Staubli VAL3: NUM.pjx

--- NUM.pjx ---
Parameters version=s7.5 stackSize=5000 millimeterUnit=true
Program file=condition.pgx
Program file=find.pgx
Program file=get.pgx
Program file=getSize.pgx
Program file=getType.pgx
Program file=isActive.pgx
Program file=load.pgx
Program file=make_if.pgx
Program file=make_NUM.pgx
Program file=onEdit.pgx
Program file=onInsert.pgx
Program file=onProgEnd.pgx
Program file=onRun.pgx
Program file=onStart.pgx
Program file=onStop.pgx
Program file=selectType.pgx
Program file=set.pgx
Program file=setValue.pgx
Data file=NUM.dtx
Library alias=use path=Disk://kernel/userPage/userPage.pjx
Library alias=cycleStatus path=Disk://cycleStatus/cycleStatus.pjx
Library alias=language path=Disk://kernel/language/language.pjx
Library alias=saveInOut path=Disk://saveInputOutput/saveInputOutput.pjx
Type name=aioItem path=Disk://kernel/template/aioItem/aioItem.pjx
Type name=countItem path=Disk://kernel/template/countItem/countItem.pjx

--- NUM.dtx ---
public string sItems
num nIndex
string sMessage
num nMode

--- condition.pgx ---
public program condition(num x_nOperator, num x_nValue, string x_sItem, bool& x_bResult)
begin
  // operator
  // <> >= > < <= ==
  x_bResult=false
  //
  switch x_nOperator
    case 0
      // <>
      if isDefined(saveInOut:cCount[x_sItem])
        x_bResult=(saveInOut:cCount[x_sItem].nCount!=x_nValue)
      elseIf isDefined(saveInOut:aCount[x_sItem])
        x_bResult=(aioGet(saveInOut:aCount[x_sItem].aAio)!=x_nValue)
      endIf
    break
    case 1
      // >=
      if isDefined(saveInOut:cCount[x_sItem])
        x_bResult=(saveInOut:cCount[x_sItem].nCount>=x_nValue)
      elseIf isDefined(saveInOut:aCount[x_sItem])
        x_bResult=(aioGet(saveInOut:aCount[x_sItem].aAio)>=x_nValue)
      endIf
    break
    case 2
      // >
      if isDefined(saveInOut:cCount[x_sItem])
        x_bResult=(saveInOut:cCount[x_sItem].nCount>x_nValue)
      elseIf isDefined(saveInOut:aCount[x_sItem])
        x_bResult=(aioGet(saveInOut:aCount[x_sItem].aAio)>x_nValue)
      endIf
    break
    case 3
      // <
      if isDefined(saveInOut:cCount[x_sItem])
        x_bResult=(saveInOut:cCount[x_sItem].nCount<x_nValue)
      elseIf isDefined(saveInOut:aCount[x_sItem])
        x_bResult=(aioGet(saveInOut:aCount[x_sItem].aAio)<x_nValue)
      endIf
    break
    case 4
      // <=
      if isDefined(saveInOut:cCount[x_sItem])
        x_bResult=(saveInOut:cCount[x_sItem].nCount<=x_nValue)
      elseIf isDefined(saveInOut:aCount[x_sItem])
        x_bResult=(aioGet(saveInOut:aCount[x_sItem].aAio)<=x_nValue)
      endIf
    break
    case 5
      // ==
      if isDefined(saveInOut:cCount[x_sItem])
        x_bResult=(saveInOut:cCount[x_sItem].nCount==x_nValue)
      elseIf isDefined(saveInOut:aCount[x_sItem])
        x_bResult=(aioGet(saveInOut:aCount[x_sItem].aAio)==x_nValue)
      endIf
    break
  endSwitch
end

--- find.pgx ---
public program find(string& x_sItem[], bool& x_bFound[])
  local num l_nIndex
  local num l_nOperator
  local num l_nValue
  local string l_sItem[2]
begin
  // REMOVE THE COUNT
  x_sItem=right(x_sItem,len(x_sItem)-len("NUM "))
  // look inside
  x_bFound=isDefined(saveInOut:cCount[x_sItem])
  if !x_bFound
    x_bFound=isDefined(saveInOut:aCount[x_sItem])
  endIf
end

--- isActive.pgx ---
public program isActive(bool& x_bActive, string x_sItem)
begin
  // check it
  if isDefined(saveInOut:cCount[x_sItem])
    x_bActive=saveInOut:cCount[x_sItem].bActive
  elseIf isDefined(saveInOut:aCount[x_sItem])
    x_bActive=(ioStatus(saveInOut:aCount[x_sItem].aAio)>=0)
  else
    // not found
    // toDO
    popUpMsg("value not found: "+x_sItem)
    x_sItem=""
  endIf
end

--- make_if.pgx ---
program make_if(string& x_sItem)
  local string l_sMessage
  local num i
  local num l_nValue
  local string l_sEmpty
  local string l_sItem
  local num l_nSizeList
  local string l_sEvent
  local bool l_bActive
  local string l_sItemList
  local num l_nKey
  local num l_nIndex
  local string l_sButton[2]
  local bool l_bYes
begin
  //
  cls()
  // Select the operator
  call language:message(l_sMessage,110)
  call use:questionDialog(l_sMessage,saveInOut:sCondition,i)
  //
  // != >= > < <= ==
  // compose the istruction
  if i>=1 and i<=size(saveInOut:sCondition)
    x_sItem=x_sItem+saveInOut:sCondition[i-1]
  else
    // escape
    x_sItem=""
    return
  endIf
  // modify the actual item
  call use:type(2,12,x_sItem)
  // insert a value
  call language:message(l_sMessage,112)
  // get the yes_no button Key
  call language:getYesNo(l_sButton)
  // ask the question
  call use:yes_no(l_sMessage,l_sButton,l_bYes)
  // check it
  if l_bYes
    //
    // reuse the operator
    //
    call saveInOut:getSize_num(l_nSizeList)
    call getType(l_sItem)
    call use:setSizeList(21,0,17,10)
    call use:listcreate(l_sItem)
    // insert in the list
    for i=0 to l_nSizeList-1
      call saveInOut:get_num(l_sItemList,i)
      call isActive(l_bActive,l_sItemList)
      if l_bActive
        call use:listadd(l_sItemList)
      endIf
    endFor
    call use:listredraw(0)
    do
      // get the key
      l_nKey=get()
      // get one input from the list
      call use:listevent(l_nKey,l_nIndex,l_sEvent)
      if l_nKey==255
        return
      endIf
    until l_nKey==270
    // check if an item has been selected
    if l_sEvent==""
      x_sItem=""
      return
    else
      x_sItem=x_sItem+"NUM "+ l_sEvent
    endIf
  else
    // use a value
    call use:changeValue(l_nValue,-10000,10000,2+len(x_sItem),12,l_sEmpty)
    x_sItem=x_sItem+toString("",l_nValue)
  endIf
  // validate
  if use:bUseEscape
    x_sItem=""
  endIf
end

--- make_NUM.pgx ---
program make_NUM(string& x_sItem)
  local string l_sMessage
  local num i
  local num l_nValue
  local string l_sEmpty
  local string l_sItem
begin
  cls()
  //
  // = =NUM +1 -1
  //
  // display the actual item
  call use:type(2,12,x_sItem)
  // Select the operator
  call language:message(l_sMessage,110)
  call use:questionDialog(l_sMessage,saveInOut:sOperator,i)
  if i!=-1
    // compose the istruction
    call use:type(2,12,x_sItem+saveInOut:sOperator[i-1])
    // modify the value
    if i==1
      // modify the actual item
      call language:message(l_sMessage,111)
      call use:changeValue(l_nValue,-10000,10000,4+len(x_sItem),12,l_sEmpty)
      x_sItem=x_sItem+saveInOut:sOperator[i-1]+toString("",l_nValue)
    elseIf i==2
      // select a new value
      call selectType(l_sItem)
      if l_sItem!=""
        x_sItem=x_sItem+"=NUM "+l_sItem
      else
        x_sItem=""
      endIf
    elseIf i>2
      // use the + - 1
      x_sItem=x_sItem+saveInOut:sOperator[i-1]
    else
      // escape -> return
    endIf
  endIf
  // validate
  if use:bUseEscape
    x_sItem=""
  endIf
end

--- onEdit.pgx ---
public program onEdit(string& x_sItem[])
  local num l_nX
  local num l_nY
  local num l_nDelay
  local bool l_bValide
  local num l_nIndex
  local num l_nOperator
  local num l_nValue
  local string l_sType
  local string l_sName
begin
  // decompose it
  call saveInOut:decompose_num(x_sItem,l_sName,l_nOperator,l_nValue)
  if l_sName!=""
    // get the item
    call saveInOut:get_num(x_sItem,l_nIndex)
    // edit it
    call make_NUM(x_sItem)
  else
    x_sItem=""
  endIf
end

--- onInsert.pgx ---
public program onInsert(string& x_sItem[])
  local string l_sEvent
begin
  cls()
  call selectType(l_sEvent)
  // exit
  if l_sEvent==""
    x_sItem=""
    return
  endIf
  //
  if x_sItem!="IF"
    // compose the instruction
    call make_NUM(l_sEvent)
  else
    // usine an IF
    call make_if(l_sEvent)
  endIf
  // update
  x_sItem=l_sEvent
end

--- onRun.pgx ---
public program onRun(string& x_sItem[])
  local num l_nValue
  local bool l_bOk
  local num l_nIndex
  local num l_nOperator
  local string l_sName
begin
  //
  // decompose
  //
  call saveInOut:decompose_num(x_sItem,l_sName,l_nOperator,l_nValue)
  //
  if l_sName!=""
    // execute
    switch l_nOperator
      case 0,1
        // =
        call setValue(l_nValue,l_sName)
      break
      case 2
        // +1
        call saveInOut:getValue_num(l_nValue,l_sName)
        l_nValue=l_nValue+1
        call setValue(l_nValue,l_sName)
      break
      case 3
        // -1
        call saveInOut:getValue_num(l_nValue,l_sName)
        l_nValue=l_nValue-1
        call setValue(l_nValue,l_sName)
      break
    endSwitch
  endIf
end

--- onStart.pgx ---
public program onStart(string& x_sItem[])
begin
  //
  // ANALOGIC VALUE
  //
  // default use the COUNTER
  call saveInOut:setOutput(10)
  call saveInOut:setInput(10)
  // MODBUS
  call saveInOut:setOutput(11)
  call saveInOut:setInput(11)
  // USER
  call saveInOut:setOutput(12)
  call saveInOut:setInput(12)
  // REMIO
  call saveInOut:setOutput(13)
  call saveInOut:setInput(13)
  // Other
  call saveInOut:setOutput(14)
  call saveInOut:setInput(14)
end

--- selectType.pgx ---
program selectType(string& x_sItem)
  local num l_nSizeList
  local string l_sItem
  local bool l_bActive
  local string l_sItemList
  local string l_sMessage
  local num l_nKey
  local string l_sEvent
  local num l_nSize
  local num i
  local string l_sName
begin
  // NUM
  call saveInOut:getSize_num(l_nSizeList)
  call getType(l_sItem)
  l_nSize=0
  //
  // create the list
  //
  call use:setSizeList(19,0,19,11)
  call use:listcreate(l_sItem)
  // insert in the list
  for i=0 to l_nSizeList-1
    call saveInOut:get_num(l_sItemList,i)
    call isActive(l_bActive,l_sItemList)
    if l_bActive
      call saveInOut:get_num(l_sItemList,i)
      call saveInOut:getItem_num(l_sName,l_sItemList)
      l_sItemList=l_sItemList+" {"+l_sName+"}"
      call use:listadd(l_sItemList)
    endIf
  endFor
  call use:selectNewField(nIndex,nIndex,0)
  call use:clear(0,13)
  call language:message(l_sMessage,63)
  call use:typeCenter(13,l_sMessage,40,true)
  do
    // get the key
    l_nKey=get()
    // get one input from the list
    call use:listevent(l_nKey,nIndex,l_sEvent)
    if l_nKey==255
      return
    endIf
  until l_nKey==270
  // save it
  if l_sEvent!=""
    x_sItem=left(l_sEvent,find(l_sEvent,"{")-1)
  else
    x_sItem=""
  endIf
end

--- set.pgx ---
public program set(string x_sName, string x_sItem)
begin
  // Get IT
  //  sName[x_nIndex]=x_sItem
  if isDefined(saveInOut:cCount[x_sItem])
    saveInOut:cCount[x_sItem].sName=x_sName
  elseIf isDefined(saveInOut:aCount[x_sItem])
    saveInOut:aCount[x_sItem].sName=x_sName
  else
    // not found
    // toDO
    popUpMsg("value not found: "+x_sItem)
    x_sItem=""
  endIf
end

--- setValue.pgx ---
public program setValue(num& x_nValue[], string x_sItem)
begin
  if find(x_sItem,"In")==-1
    // set the data only for output
    if isDefined(saveInOut:cCount[x_sItem])
      saveInOut:cCount[x_sItem].nCount=x_nValue
    elseIf isDefined(saveInOut:aCount[x_sItem])
      aioSet(saveInOut:aCount[x_sItem].aAio,x_nValue)
    endIf
  endIf
end
